// TwinCAT 3 PLC project ProjectB
// ProgramVersion: 3.1.4022.7
// libraries:
//   LCLS General, * (SLAC)
//   Tc2_Standard, * (Beckhoff Automation GmbH)
//   Tc2_System, * (Beckhoff Automation GmbH)
//   Tc3_Module, * (Beckhoff Automation GmbH)
// project tree:
//   DUTs/ ST_ProjectB.TcDUT
//   GVLs/ GVL_ProjectB.TcGVL
//   / PlcTask.TcTTO
//   POUs/ MAIN.TcPOU
// real-time tasks:
//   TASK PlcTask: cycle T#10ms, priority 20, ADS port 350

CONFIGURATION ProjectB
    RESOURCE PLC ON TwinCAT3
        TASK PlcTask(INTERVAL := T#10ms, PRIORITY := 20);
        PROGRAM MAIN WITH PlcTask : MAIN;
    END_RESOURCE
END_CONFIGURATION

// ---- DUTs/ST_ProjectB.TcDUT
TYPE ST_ProjectB :
STRUCT
	iProjectB : INT;
END_STRUCT
END_TYPE

// ---- GVLs/GVL_ProjectB.TcGVL
{attribute 'qualified_only'}
VAR_GLOBAL
	bProjectB : BOOL;
END_VAR

// ---- POUs/MAIN.TcPOU
PROGRAM MAIN
VAR
	bProjectB : BOOL;
	fbLogger : FB_LogHandler;
END_VAR

fbLogger();

END_PROGRAM
